INTERFACE I_AdsChannel EXTENDS I_Channel

PROPERTY PUBLIC P_NetID : STRING
GET
END_GET
END_PROPERTY

PROPERTY PUBLIC P_Port : UINT
GET
END_GET
END_PROPERTY

END_INTERFACE

(* stored: Version 1.1.0.1
   Itf I_AdsChannel: Id {64432f8c-0ebd-0faf-174b-858c109f0548}
   Property P_NetID: Id {a4279ce0-81fa-0631-33ce-f382c94ec314}
   Get Get: Id {1f93eb45-4981-0222-1e91-5abf9c3b4cdd}
   Property P_Port: Id {aba33edd-ad89-0a11-3f51-37400193d214}
   Get Get: Id {0c1a6525-84a6-0e7a-19b2-850a8c8a4395} *)
